(* PLC project AtoB, Unknown Unnamed 1 *)
(* stored: creationDateTime 2020-12-12T16:27:35, modificationDateTime 2020-12-12T20:24:46 *)

PROGRAM AtoB
  VAR
    StartButton AT %IX100.0 : BOOL;
    Sensor AT %IX100.1 : BOOL;
    Conveyor AT %QX100.0 : BOOL;
  END_VAR

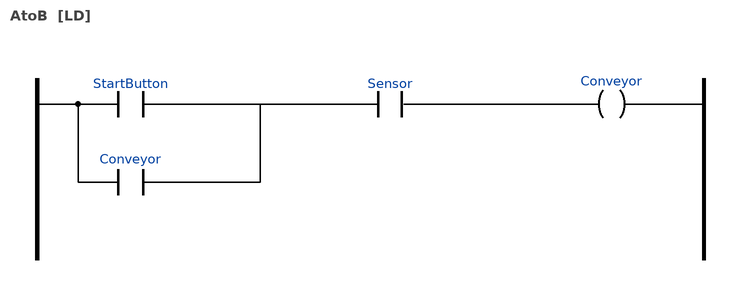
(* LD diagram, written out as Structured Text *)
Conveyor := (StartButton OR Conveyor) AND Sensor;
END_PROGRAM

CONFIGURATION Config0
  RESOURCE Res0 ON PLC
    TASK task0(INTERVAL := T#20ms, PRIORITY := 0);
    PROGRAM instance0 WITH task0 : AtoB;
  END_RESOURCE
END_CONFIGURATION
